FUNCTION_BLOCK Station001ProcessData
VAR_INPUT
END_VAR
VAR_OUTPUT
END_VAR
VAR
END_VAR

END_FUNCTION_BLOCK

(* stored: Version 1.1.0.1, ProductVersion 3.1.4024.9
   POU Station001ProcessData: Id {73945634-36d0-4813-8f9d-01a731012014}, SpecialFunc None *)
